DATA_BLOCK "DB_群控状态"
{ S7_Optimized_Access := 'TRUE' }
VERSION : 0.1
NON_RETAIN
   VAR
      外呼上已登记 : Array[1..9] of Bool;
      外呼下已登记 : Array[2..10] of Bool;
      外呼上分配给梯号 : Array[1..9] of Int;
      外呼下分配给梯号 : Array[2..10] of Int;
      梯当前楼层 : Array[1..3] of Int;
      梯运行方向 : Array[1..3] of Int;
      梯是否服务中 : Array[1..3] of Bool;
      梯是否故障 : Array[1..3] of Bool;
      梯是否满载 : Array[1..3] of Bool;
      群控扫描计数器 : Int;
      外呼上等待周期 : Array[1..9] of Int;
      外呼下等待周期 : Array[2..10] of Int;
      梯是否检修 : Array[1..3] of Bool;
      检修退出屏蔽计数 : Array[1..3] of Int;   // 检修信号0->1或1->0后继续屏蔸运动输出，50扫描周期约500ms
      检修上次有效 : Array[1..3] of Bool;   // 上一扫描周期检修信号，用于检测0->1/1->0边沿
   END_VAR


BEGIN

END_DATA_BLOCK

